PROGRAM AnyTypeHelper

METHOD GetAnyDescriptorByVariable : __SYSTEM.AnyType
VAR_INPUT
	variable : ANY;
END_VAR
GetAnyDescriptorByVariable := variable;
END_METHOD

END_PROGRAM

(* stored: Version 1.1.0.1
   POU AnyTypeHelper: Id {30a9a158-f31f-4666-9b77-4b974af8545f}, SpecialFunc None
   Method GetAnyDescriptorByVariable: Id {1d943783-b113-4944-ae42-a6c966c7d38f} *)
